FUNCTION_BLOCK ColorDebug (* Basic Function Block Type *)
  (* Standard: 61499-2 *)
  (* Version 0.0, 22/06/2022, Lernfabrik, WBK hackaton, Template *)
  PACKAGE Main;
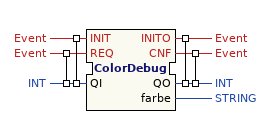
  EVENT_INPUT
    INIT WITH QI; (* Initialization Request *)
    REQ WITH QI; (* Normal Execution Request *)
  END_EVENT
  EVENT_OUTPUT
    INITO WITH QO; (* Initialization Confirm *)
    CNF WITH QO; (* Execution Confirmation *)
  END_EVENT
  VAR_INPUT
    QI : INT; (* Input event qualifier *)
  END_VAR
  VAR_OUTPUT
    QO : INT; (* Output event qualifier *)
    farbe : STRING; (* olo *)
  END_VAR
  VAR
    Minimum : INT;
  END_VAR
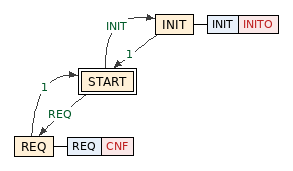
  EC_STATES
    START; (* Initial State *)
    INIT : INIT -> INITO; (* Initialization *)
    REQ : REQ -> CNF; (* Normal execution *)
  END_STATES
  EC_TRANSITIONS
    START TO INIT := INIT;
    INIT TO START := 1;
    START TO REQ := REQ;
    REQ TO START := 1;
  END_TRANSITIONS
  ALGORITHM INIT IN ST: (* Initialization algorithm *)
Minimum := 32000;
QO := Minimum;
  END_ALGORITHM
  ALGORITHM REQ IN ST: (* Normally executed algorithm *)
IF QI < Minimum THEN
Minimum := QI;
END_IF;
QO := Minimum;

farbe := 'NONE';

IF  QI <20300
THEN
farbe := 'WEISS';
END_IF;

IF  QI > 20850 AND QI <21450
THEN
farbe := 'ROT';
END_IF;

IF  QI > 26650 AND QI < 27300
THEN
farbe := 'BLAU';
END_IF;
  END_ALGORITHM
END_FUNCTION_BLOCK
